  STRUCT
   FC1_SEND_1 : ARRAY  [0 .. 699 ] OF BYTE  := B#16#0;
  END_STRUCT ;
BEGIN
   FC1_SEND_1[0] := B#16#0;
   FC1_SEND_1[1] := B#16#0;
   FC1_SEND_1[2] := B#16#0;
   FC1_SEND_1[3] := B#16#0;
   FC1_SEND_1[4] := B#16#0;
   FC1_SEND_1[5] := B#16#0;
   FC1_SEND_1[6] := B#16#0;
   FC1_SEND_1[7] := B#16#0;
   FC1_SEND_1[8] := B#16#0;
   FC1_SEND_1[9] := B#16#0;
   FC1_SEND_1[10] := B#16#0;
   FC1_SEND_1[11] := B#16#0;
   FC1_SEND_1[12] := B#16#0;
   FC1_SEND_1[13] := B#16#0;
   FC1_SEND_1[14] := B#16#0;
   FC1_SEND_1[15] := B#16#0;
   FC1_SEND_1[16] := B#16#0;
   FC1_SEND_1[17] := B#16#0;
   FC1_SEND_1[18] := B#16#0;
   FC1_SEND_1[19] := B#16#0;
   FC1_SEND_1[20] := B#16#0;
   FC1_SEND_1[21] := B#16#0;
   FC1_SEND_1[22] := B#16#0;
   FC1_SEND_1[23] := B#16#0;
   FC1_SEND_1[24] := B#16#0;
   FC1_SEND_1[25] := B#16#0;
   FC1_SEND_1[26] := B#16#0;
   FC1_SEND_1[27] := B#16#0;
   FC1_SEND_1[28] := B#16#0;
   FC1_SEND_1[29] := B#16#0;
   FC1_SEND_1[30] := B#16#0;
   FC1_SEND_1[31] := B#16#0;
   FC1_SEND_1[32] := B#16#0;
   FC1_SEND_1[33] := B#16#0;
   FC1_SEND_1[34] := B#16#0;
   FC1_SEND_1[35] := B#16#0;
   FC1_SEND_1[36] := B#16#0;
   FC1_SEND_1[37] := B#16#0;
   FC1_SEND_1[38] := B#16#0;
   FC1_SEND_1[39] := B#16#0;
   FC1_SEND_1[40] := B#16#0;
   FC1_SEND_1[41] := B#16#0;
   FC1_SEND_1[42] := B#16#0;
   FC1_SEND_1[43] := B#16#0;
   FC1_SEND_1[44] := B#16#0;
   FC1_SEND_1[45] := B#16#0;
   FC1_SEND_1[46] := B#16#0;
   FC1_SEND_1[47] := B#16#0;
   FC1_SEND_1[48] := B#16#0;
   FC1_SEND_1[49] := B#16#0;
   FC1_SEND_1[50] := B#16#0;
   FC1_SEND_1[51] := B#16#0;
   FC1_SEND_1[52] := B#16#0;
   FC1_SEND_1[53] := B#16#0;
   FC1_SEND_1[54] := B#16#0;
   FC1_SEND_1[55] := B#16#0;
   FC1_SEND_1[56] := B#16#0;
   FC1_SEND_1[57] := B#16#0;
   FC1_SEND_1[58] := B#16#0;
   FC1_SEND_1[59] := B#16#0;
   FC1_SEND_1[60] := B#16#0;
   FC1_SEND_1[61] := B#16#0;
   FC1_SEND_1[62] := B#16#0;
   FC1_SEND_1[63] := B#16#0;
   FC1_SEND_1[64] := B#16#0;
   FC1_SEND_1[65] := B#16#0;
   FC1_SEND_1[66] := B#16#0;
   FC1_SEND_1[67] := B#16#0;
   FC1_SEND_1[68] := B#16#0;
   FC1_SEND_1[69] := B#16#0;
   FC1_SEND_1[70] := B#16#0;
   FC1_SEND_1[71] := B#16#0;
   FC1_SEND_1[72] := B#16#0;
   FC1_SEND_1[73] := B#16#0;
   FC1_SEND_1[74] := B#16#0;
   FC1_SEND_1[75] := B#16#0;
   FC1_SEND_1[76] := B#16#0;
   FC1_SEND_1[77] := B#16#0;
   FC1_SEND_1[78] := B#16#0;
   FC1_SEND_1[79] := B#16#0;
   FC1_SEND_1[80] := B#16#0;
   FC1_SEND_1[81] := B#16#0;
   FC1_SEND_1[82] := B#16#0;
   FC1_SEND_1[83] := B#16#0;
   FC1_SEND_1[84] := B#16#0;
   FC1_SEND_1[85] := B#16#0;
   FC1_SEND_1[86] := B#16#0;
   FC1_SEND_1[87] := B#16#0;
   FC1_SEND_1[88] := B#16#0;
   FC1_SEND_1[89] := B#16#0;
   FC1_SEND_1[90] := B#16#0;
   FC1_SEND_1[91] := B#16#0;
   FC1_SEND_1[92] := B#16#0;
   FC1_SEND_1[93] := B#16#0;
   FC1_SEND_1[94] := B#16#0;
   FC1_SEND_1[95] := B#16#0;
   FC1_SEND_1[96] := B#16#0;
   FC1_SEND_1[97] := B#16#0;
   FC1_SEND_1[98] := B#16#0;
   FC1_SEND_1[99] := B#16#0;
   FC1_SEND_1[100] := B#16#0;
   FC1_SEND_1[101] := B#16#0;
   FC1_SEND_1[102] := B#16#0;
   FC1_SEND_1[103] := B#16#0;
   FC1_SEND_1[104] := B#16#0;
   FC1_SEND_1[105] := B#16#0;
   FC1_SEND_1[106] := B#16#0;
   FC1_SEND_1[107] := B#16#0;
   FC1_SEND_1[108] := B#16#0;
   FC1_SEND_1[109] := B#16#0;
   FC1_SEND_1[110] := B#16#0;
   FC1_SEND_1[111] := B#16#0;
   FC1_SEND_1[112] := B#16#0;
   FC1_SEND_1[113] := B#16#0;
   FC1_SEND_1[114] := B#16#0;
   FC1_SEND_1[115] := B#16#0;
   FC1_SEND_1[116] := B#16#0;
   FC1_SEND_1[117] := B#16#0;
   FC1_SEND_1[118] := B#16#0;
   FC1_SEND_1[119] := B#16#0;
   FC1_SEND_1[120] := B#16#0;
   FC1_SEND_1[121] := B#16#0;
   FC1_SEND_1[122] := B#16#0;
   FC1_SEND_1[123] := B#16#0;
   FC1_SEND_1[124] := B#16#0;
   FC1_SEND_1[125] := B#16#0;
   FC1_SEND_1[126] := B#16#0;
   FC1_SEND_1[127] := B#16#0;
   FC1_SEND_1[128] := B#16#0;
   FC1_SEND_1[129] := B#16#0;
   FC1_SEND_1[130] := B#16#0;
   FC1_SEND_1[131] := B#16#0;
   FC1_SEND_1[132] := B#16#0;
   FC1_SEND_1[133] := B#16#0;
   FC1_SEND_1[134] := B#16#0;
   FC1_SEND_1[135] := B#16#0;
   FC1_SEND_1[136] := B#16#0;
   FC1_SEND_1[137] := B#16#0;
   FC1_SEND_1[138] := B#16#0;
   FC1_SEND_1[139] := B#16#0;
   FC1_SEND_1[140] := B#16#0;
   FC1_SEND_1[141] := B#16#0;
   FC1_SEND_1[142] := B#16#0;
   FC1_SEND_1[143] := B#16#0;
   FC1_SEND_1[144] := B#16#0;
   FC1_SEND_1[145] := B#16#0;
   FC1_SEND_1[146] := B#16#0;
   FC1_SEND_1[147] := B#16#0;
   FC1_SEND_1[148] := B#16#0;
   FC1_SEND_1[149] := B#16#0;
   FC1_SEND_1[150] := B#16#0;
   FC1_SEND_1[151] := B#16#0;
   FC1_SEND_1[152] := B#16#0;
   FC1_SEND_1[153] := B#16#0;
   FC1_SEND_1[154] := B#16#0;
   FC1_SEND_1[155] := B#16#0;
   FC1_SEND_1[156] := B#16#0;
   FC1_SEND_1[157] := B#16#0;
   FC1_SEND_1[158] := B#16#0;
   FC1_SEND_1[159] := B#16#0;
   FC1_SEND_1[160] := B#16#0;
   FC1_SEND_1[161] := B#16#0;
   FC1_SEND_1[162] := B#16#0;
   FC1_SEND_1[163] := B#16#0;
   FC1_SEND_1[164] := B#16#0;
   FC1_SEND_1[165] := B#16#0;
   FC1_SEND_1[166] := B#16#0;
   FC1_SEND_1[167] := B#16#0;
   FC1_SEND_1[168] := B#16#0;
   FC1_SEND_1[169] := B#16#0;
   FC1_SEND_1[170] := B#16#0;
   FC1_SEND_1[171] := B#16#0;
   FC1_SEND_1[172] := B#16#0;
   FC1_SEND_1[173] := B#16#0;
   FC1_SEND_1[174] := B#16#0;
   FC1_SEND_1[175] := B#16#0;
   FC1_SEND_1[176] := B#16#0;
   FC1_SEND_1[177] := B#16#0;
   FC1_SEND_1[178] := B#16#0;
   FC1_SEND_1[179] := B#16#0;
   FC1_SEND_1[180] := B#16#0;
   FC1_SEND_1[181] := B#16#0;
   FC1_SEND_1[182] := B#16#0;
   FC1_SEND_1[183] := B#16#0;
   FC1_SEND_1[184] := B#16#0;
   FC1_SEND_1[185] := B#16#0;
   FC1_SEND_1[186] := B#16#0;
   FC1_SEND_1[187] := B#16#0;
   FC1_SEND_1[188] := B#16#0;
   FC1_SEND_1[189] := B#16#0;
   FC1_SEND_1[190] := B#16#0;
   FC1_SEND_1[191] := B#16#0;
   FC1_SEND_1[192] := B#16#0;
   FC1_SEND_1[193] := B#16#0;
   FC1_SEND_1[194] := B#16#0;
   FC1_SEND_1[195] := B#16#0;
   FC1_SEND_1[196] := B#16#0;
   FC1_SEND_1[197] := B#16#0;
   FC1_SEND_1[198] := B#16#0;
   FC1_SEND_1[199] := B#16#0;
   FC1_SEND_1[200] := B#16#0;
   FC1_SEND_1[201] := B#16#0;
   FC1_SEND_1[202] := B#16#0;
   FC1_SEND_1[203] := B#16#0;
   FC1_SEND_1[204] := B#16#0;
   FC1_SEND_1[205] := B#16#0;
   FC1_SEND_1[206] := B#16#0;
   FC1_SEND_1[207] := B#16#0;
   FC1_SEND_1[208] := B#16#0;
   FC1_SEND_1[209] := B#16#0;
   FC1_SEND_1[210] := B#16#0;
   FC1_SEND_1[211] := B#16#0;
   FC1_SEND_1[212] := B#16#0;
   FC1_SEND_1[213] := B#16#0;
   FC1_SEND_1[214] := B#16#0;
   FC1_SEND_1[215] := B#16#0;
   FC1_SEND_1[216] := B#16#0;
   FC1_SEND_1[217] := B#16#0;
   FC1_SEND_1[218] := B#16#0;
   FC1_SEND_1[219] := B#16#0;
   FC1_SEND_1[220] := B#16#0;
   FC1_SEND_1[221] := B#16#0;
   FC1_SEND_1[222] := B#16#0;
   FC1_SEND_1[223] := B#16#0;
   FC1_SEND_1[224] := B#16#0;
   FC1_SEND_1[225] := B#16#0;
   FC1_SEND_1[226] := B#16#0;
   FC1_SEND_1[227] := B#16#0;
   FC1_SEND_1[228] := B#16#0;
   FC1_SEND_1[229] := B#16#0;
   FC1_SEND_1[230] := B#16#0;
   FC1_SEND_1[231] := B#16#0;
   FC1_SEND_1[232] := B#16#0;
   FC1_SEND_1[233] := B#16#0;
   FC1_SEND_1[234] := B#16#0;
   FC1_SEND_1[235] := B#16#0;
   FC1_SEND_1[236] := B#16#0;
   FC1_SEND_1[237] := B#16#0;
   FC1_SEND_1[238] := B#16#0;
   FC1_SEND_1[239] := B#16#0;
   FC1_SEND_1[240] := B#16#0;
   FC1_SEND_1[241] := B#16#0;
   FC1_SEND_1[242] := B#16#0;
   FC1_SEND_1[243] := B#16#0;
   FC1_SEND_1[244] := B#16#0;
   FC1_SEND_1[245] := B#16#0;
   FC1_SEND_1[246] := B#16#0;
   FC1_SEND_1[247] := B#16#0;
   FC1_SEND_1[248] := B#16#0;
   FC1_SEND_1[249] := B#16#0;
   FC1_SEND_1[250] := B#16#0;
   FC1_SEND_1[251] := B#16#0;
   FC1_SEND_1[252] := B#16#0;
   FC1_SEND_1[253] := B#16#0;
   FC1_SEND_1[254] := B#16#0;
   FC1_SEND_1[255] := B#16#0;
   FC1_SEND_1[256] := B#16#0;
   FC1_SEND_1[257] := B#16#0;
   FC1_SEND_1[258] := B#16#0;
   FC1_SEND_1[259] := B#16#0;
   FC1_SEND_1[260] := B#16#0;
   FC1_SEND_1[261] := B#16#0;
   FC1_SEND_1[262] := B#16#0;
   FC1_SEND_1[263] := B#16#0;
   FC1_SEND_1[264] := B#16#0;
   FC1_SEND_1[265] := B#16#0;
   FC1_SEND_1[266] := B#16#0;
   FC1_SEND_1[267] := B#16#0;
   FC1_SEND_1[268] := B#16#0;
   FC1_SEND_1[269] := B#16#0;
   FC1_SEND_1[270] := B#16#0;
   FC1_SEND_1[271] := B#16#0;
   FC1_SEND_1[272] := B#16#0;
   FC1_SEND_1[273] := B#16#0;
   FC1_SEND_1[274] := B#16#0;
   FC1_SEND_1[275] := B#16#0;
   FC1_SEND_1[276] := B#16#0;
   FC1_SEND_1[277] := B#16#0;
   FC1_SEND_1[278] := B#16#0;
   FC1_SEND_1[279] := B#16#0;
   FC1_SEND_1[280] := B#16#0;
   FC1_SEND_1[281] := B#16#0;
   FC1_SEND_1[282] := B#16#0;
   FC1_SEND_1[283] := B#16#0;
   FC1_SEND_1[284] := B#16#0;
   FC1_SEND_1[285] := B#16#0;
   FC1_SEND_1[286] := B#16#0;
   FC1_SEND_1[287] := B#16#0;
   FC1_SEND_1[288] := B#16#0;
   FC1_SEND_1[289] := B#16#0;
   FC1_SEND_1[290] := B#16#0;
   FC1_SEND_1[291] := B#16#0;
   FC1_SEND_1[292] := B#16#0;
   FC1_SEND_1[293] := B#16#0;
   FC1_SEND_1[294] := B#16#0;
   FC1_SEND_1[295] := B#16#0;
   FC1_SEND_1[296] := B#16#0;
   FC1_SEND_1[297] := B#16#0;
   FC1_SEND_1[298] := B#16#0;
   FC1_SEND_1[299] := B#16#0;
   FC1_SEND_1[300] := B#16#0;
   FC1_SEND_1[301] := B#16#0;
   FC1_SEND_1[302] := B#16#0;
   FC1_SEND_1[303] := B#16#0;
   FC1_SEND_1[304] := B#16#0;
   FC1_SEND_1[305] := B#16#0;
   FC1_SEND_1[306] := B#16#0;
   FC1_SEND_1[307] := B#16#0;
   FC1_SEND_1[308] := B#16#0;
   FC1_SEND_1[309] := B#16#0;
   FC1_SEND_1[310] := B#16#0;
   FC1_SEND_1[311] := B#16#0;
   FC1_SEND_1[312] := B#16#0;
   FC1_SEND_1[313] := B#16#0;
   FC1_SEND_1[314] := B#16#0;
   FC1_SEND_1[315] := B#16#0;
   FC1_SEND_1[316] := B#16#0;
   FC1_SEND_1[317] := B#16#0;
   FC1_SEND_1[318] := B#16#0;
   FC1_SEND_1[319] := B#16#0;
   FC1_SEND_1[320] := B#16#0;
   FC1_SEND_1[321] := B#16#0;
   FC1_SEND_1[322] := B#16#0;
   FC1_SEND_1[323] := B#16#0;
   FC1_SEND_1[324] := B#16#0;
   FC1_SEND_1[325] := B#16#0;
   FC1_SEND_1[326] := B#16#0;
   FC1_SEND_1[327] := B#16#0;
   FC1_SEND_1[328] := B#16#0;
   FC1_SEND_1[329] := B#16#0;
   FC1_SEND_1[330] := B#16#0;
   FC1_SEND_1[331] := B#16#0;
   FC1_SEND_1[332] := B#16#0;
   FC1_SEND_1[333] := B#16#0;
   FC1_SEND_1[334] := B#16#0;
   FC1_SEND_1[335] := B#16#0;
   FC1_SEND_1[336] := B#16#0;
   FC1_SEND_1[337] := B#16#0;
   FC1_SEND_1[338] := B#16#0;
   FC1_SEND_1[339] := B#16#0;
   FC1_SEND_1[340] := B#16#0;
   FC1_SEND_1[341] := B#16#0;
   FC1_SEND_1[342] := B#16#0;
   FC1_SEND_1[343] := B#16#0;
   FC1_SEND_1[344] := B#16#0;
   FC1_SEND_1[345] := B#16#0;
   FC1_SEND_1[346] := B#16#0;
   FC1_SEND_1[347] := B#16#0;
   FC1_SEND_1[348] := B#16#0;
   FC1_SEND_1[349] := B#16#0;
   FC1_SEND_1[350] := B#16#0;
   FC1_SEND_1[351] := B#16#0;
   FC1_SEND_1[352] := B#16#0;
   FC1_SEND_1[353] := B#16#0;
   FC1_SEND_1[354] := B#16#0;
   FC1_SEND_1[355] := B#16#0;
   FC1_SEND_1[356] := B#16#0;
   FC1_SEND_1[357] := B#16#0;
   FC1_SEND_1[358] := B#16#0;
   FC1_SEND_1[359] := B#16#0;
   FC1_SEND_1[360] := B#16#0;
   FC1_SEND_1[361] := B#16#0;
   FC1_SEND_1[362] := B#16#0;
   FC1_SEND_1[363] := B#16#0;
   FC1_SEND_1[364] := B#16#0;
   FC1_SEND_1[365] := B#16#0;
   FC1_SEND_1[366] := B#16#0;
   FC1_SEND_1[367] := B#16#0;
   FC1_SEND_1[368] := B#16#0;
   FC1_SEND_1[369] := B#16#0;
   FC1_SEND_1[370] := B#16#0;
   FC1_SEND_1[371] := B#16#0;
   FC1_SEND_1[372] := B#16#0;
   FC1_SEND_1[373] := B#16#0;
   FC1_SEND_1[374] := B#16#0;
   FC1_SEND_1[375] := B#16#0;
   FC1_SEND_1[376] := B#16#0;
   FC1_SEND_1[377] := B#16#0;
   FC1_SEND_1[378] := B#16#0;
   FC1_SEND_1[379] := B#16#0;
   FC1_SEND_1[380] := B#16#0;
   FC1_SEND_1[381] := B#16#0;
   FC1_SEND_1[382] := B#16#0;
   FC1_SEND_1[383] := B#16#0;
   FC1_SEND_1[384] := B#16#0;
   FC1_SEND_1[385] := B#16#0;
   FC1_SEND_1[386] := B#16#0;
   FC1_SEND_1[387] := B#16#0;
   FC1_SEND_1[388] := B#16#0;
   FC1_SEND_1[389] := B#16#0;
   FC1_SEND_1[390] := B#16#0;
   FC1_SEND_1[391] := B#16#0;
   FC1_SEND_1[392] := B#16#0;
   FC1_SEND_1[393] := B#16#0;
   FC1_SEND_1[394] := B#16#0;
   FC1_SEND_1[395] := B#16#0;
   FC1_SEND_1[396] := B#16#0;
   FC1_SEND_1[397] := B#16#0;
   FC1_SEND_1[398] := B#16#0;
   FC1_SEND_1[399] := B#16#0;
   FC1_SEND_1[400] := B#16#0;
   FC1_SEND_1[401] := B#16#0;
   FC1_SEND_1[402] := B#16#0;
   FC1_SEND_1[403] := B#16#0;
   FC1_SEND_1[404] := B#16#0;
   FC1_SEND_1[405] := B#16#0;
   FC1_SEND_1[406] := B#16#0;
   FC1_SEND_1[407] := B#16#0;
   FC1_SEND_1[408] := B#16#0;
   FC1_SEND_1[409] := B#16#0;
   FC1_SEND_1[410] := B#16#0;
   FC1_SEND_1[411] := B#16#0;
   FC1_SEND_1[412] := B#16#0;
   FC1_SEND_1[413] := B#16#0;
   FC1_SEND_1[414] := B#16#0;
   FC1_SEND_1[415] := B#16#0;
   FC1_SEND_1[416] := B#16#0;
   FC1_SEND_1[417] := B#16#0;
   FC1_SEND_1[418] := B#16#0;
   FC1_SEND_1[419] := B#16#0;
   FC1_SEND_1[420] := B#16#0;
   FC1_SEND_1[421] := B#16#0;
   FC1_SEND_1[422] := B#16#0;
   FC1_SEND_1[423] := B#16#0;
   FC1_SEND_1[424] := B#16#0;
   FC1_SEND_1[425] := B#16#0;
   FC1_SEND_1[426] := B#16#0;
   FC1_SEND_1[427] := B#16#0;
   FC1_SEND_1[428] := B#16#0;
   FC1_SEND_1[429] := B#16#0;
   FC1_SEND_1[430] := B#16#0;
   FC1_SEND_1[431] := B#16#0;
   FC1_SEND_1[432] := B#16#0;
   FC1_SEND_1[433] := B#16#0;
   FC1_SEND_1[434] := B#16#0;
   FC1_SEND_1[435] := B#16#0;
   FC1_SEND_1[436] := B#16#0;
   FC1_SEND_1[437] := B#16#0;
   FC1_SEND_1[438] := B#16#0;
   FC1_SEND_1[439] := B#16#0;
   FC1_SEND_1[440] := B#16#0;
   FC1_SEND_1[441] := B#16#0;
   FC1_SEND_1[442] := B#16#0;
   FC1_SEND_1[443] := B#16#0;
   FC1_SEND_1[444] := B#16#0;
   FC1_SEND_1[445] := B#16#0;
   FC1_SEND_1[446] := B#16#0;
   FC1_SEND_1[447] := B#16#0;
   FC1_SEND_1[448] := B#16#0;
   FC1_SEND_1[449] := B#16#0;
   FC1_SEND_1[450] := B#16#0;
   FC1_SEND_1[451] := B#16#0;
   FC1_SEND_1[452] := B#16#0;
   FC1_SEND_1[453] := B#16#0;
   FC1_SEND_1[454] := B#16#0;
   FC1_SEND_1[455] := B#16#0;
   FC1_SEND_1[456] := B#16#0;
   FC1_SEND_1[457] := B#16#0;
   FC1_SEND_1[458] := B#16#0;
   FC1_SEND_1[459] := B#16#0;
   FC1_SEND_1[460] := B#16#0;
   FC1_SEND_1[461] := B#16#0;
   FC1_SEND_1[462] := B#16#0;
   FC1_SEND_1[463] := B#16#0;
   FC1_SEND_1[464] := B#16#0;
   FC1_SEND_1[465] := B#16#0;
   FC1_SEND_1[466] := B#16#0;
   FC1_SEND_1[467] := B#16#0;
   FC1_SEND_1[468] := B#16#0;
   FC1_SEND_1[469] := B#16#0;
   FC1_SEND_1[470] := B#16#0;
   FC1_SEND_1[471] := B#16#0;
   FC1_SEND_1[472] := B#16#0;
   FC1_SEND_1[473] := B#16#0;
   FC1_SEND_1[474] := B#16#0;
   FC1_SEND_1[475] := B#16#0;
   FC1_SEND_1[476] := B#16#0;
   FC1_SEND_1[477] := B#16#0;
   FC1_SEND_1[478] := B#16#0;
   FC1_SEND_1[479] := B#16#0;
   FC1_SEND_1[480] := B#16#0;
   FC1_SEND_1[481] := B#16#0;
   FC1_SEND_1[482] := B#16#0;
   FC1_SEND_1[483] := B#16#0;
   FC1_SEND_1[484] := B#16#0;
   FC1_SEND_1[485] := B#16#0;
   FC1_SEND_1[486] := B#16#0;
   FC1_SEND_1[487] := B#16#0;
   FC1_SEND_1[488] := B#16#0;
   FC1_SEND_1[489] := B#16#0;
   FC1_SEND_1[490] := B#16#0;
   FC1_SEND_1[491] := B#16#0;
   FC1_SEND_1[492] := B#16#0;
   FC1_SEND_1[493] := B#16#0;
   FC1_SEND_1[494] := B#16#0;
   FC1_SEND_1[495] := B#16#0;
   FC1_SEND_1[496] := B#16#0;
   FC1_SEND_1[497] := B#16#0;
   FC1_SEND_1[498] := B#16#0;
   FC1_SEND_1[499] := B#16#0;
   FC1_SEND_1[500] := B#16#0;
   FC1_SEND_1[501] := B#16#0;
   FC1_SEND_1[502] := B#16#0;
   FC1_SEND_1[503] := B#16#0;
   FC1_SEND_1[504] := B#16#0;
   FC1_SEND_1[505] := B#16#0;
   FC1_SEND_1[506] := B#16#0;
   FC1_SEND_1[507] := B#16#0;
   FC1_SEND_1[508] := B#16#0;
   FC1_SEND_1[509] := B#16#0;
   FC1_SEND_1[510] := B#16#0;
   FC1_SEND_1[511] := B#16#0;
   FC1_SEND_1[512] := B#16#0;
   FC1_SEND_1[513] := B#16#0;
   FC1_SEND_1[514] := B#16#0;
   FC1_SEND_1[515] := B#16#0;
   FC1_SEND_1[516] := B#16#0;
   FC1_SEND_1[517] := B#16#0;
   FC1_SEND_1[518] := B#16#0;
   FC1_SEND_1[519] := B#16#0;
   FC1_SEND_1[520] := B#16#0;
   FC1_SEND_1[521] := B#16#0;
   FC1_SEND_1[522] := B#16#0;
   FC1_SEND_1[523] := B#16#0;
   FC1_SEND_1[524] := B#16#0;
   FC1_SEND_1[525] := B#16#0;
   FC1_SEND_1[526] := B#16#0;
   FC1_SEND_1[527] := B#16#0;
   FC1_SEND_1[528] := B#16#0;
   FC1_SEND_1[529] := B#16#0;
   FC1_SEND_1[530] := B#16#0;
   FC1_SEND_1[531] := B#16#0;
   FC1_SEND_1[532] := B#16#0;
   FC1_SEND_1[533] := B#16#0;
   FC1_SEND_1[534] := B#16#0;
   FC1_SEND_1[535] := B#16#0;
   FC1_SEND_1[536] := B#16#0;
   FC1_SEND_1[537] := B#16#0;
   FC1_SEND_1[538] := B#16#0;
   FC1_SEND_1[539] := B#16#0;
   FC1_SEND_1[540] := B#16#0;
   FC1_SEND_1[541] := B#16#0;
   FC1_SEND_1[542] := B#16#0;
   FC1_SEND_1[543] := B#16#0;
   FC1_SEND_1[544] := B#16#0;
   FC1_SEND_1[545] := B#16#0;
   FC1_SEND_1[546] := B#16#0;
   FC1_SEND_1[547] := B#16#0;
   FC1_SEND_1[548] := B#16#0;
   FC1_SEND_1[549] := B#16#0;
   FC1_SEND_1[550] := B#16#0;
   FC1_SEND_1[551] := B#16#0;
   FC1_SEND_1[552] := B#16#0;
   FC1_SEND_1[553] := B#16#0;
   FC1_SEND_1[554] := B#16#0;
   FC1_SEND_1[555] := B#16#0;
   FC1_SEND_1[556] := B#16#0;
   FC1_SEND_1[557] := B#16#0;
   FC1_SEND_1[558] := B#16#0;
   FC1_SEND_1[559] := B#16#0;
   FC1_SEND_1[560] := B#16#0;
   FC1_SEND_1[561] := B#16#0;
   FC1_SEND_1[562] := B#16#0;
   FC1_SEND_1[563] := B#16#0;
   FC1_SEND_1[564] := B#16#0;
   FC1_SEND_1[565] := B#16#0;
   FC1_SEND_1[566] := B#16#0;
   FC1_SEND_1[567] := B#16#0;
   FC1_SEND_1[568] := B#16#0;
   FC1_SEND_1[569] := B#16#0;
   FC1_SEND_1[570] := B#16#0;
   FC1_SEND_1[571] := B#16#0;
   FC1_SEND_1[572] := B#16#0;
   FC1_SEND_1[573] := B#16#0;
   FC1_SEND_1[574] := B#16#0;
   FC1_SEND_1[575] := B#16#0;
   FC1_SEND_1[576] := B#16#0;
   FC1_SEND_1[577] := B#16#0;
   FC1_SEND_1[578] := B#16#0;
   FC1_SEND_1[579] := B#16#0;
   FC1_SEND_1[580] := B#16#0;
   FC1_SEND_1[581] := B#16#0;
   FC1_SEND_1[582] := B#16#0;
   FC1_SEND_1[583] := B#16#0;
   FC1_SEND_1[584] := B#16#0;
   FC1_SEND_1[585] := B#16#0;
   FC1_SEND_1[586] := B#16#0;
   FC1_SEND_1[587] := B#16#0;
   FC1_SEND_1[588] := B#16#0;
   FC1_SEND_1[589] := B#16#0;
   FC1_SEND_1[590] := B#16#0;
   FC1_SEND_1[591] := B#16#0;
   FC1_SEND_1[592] := B#16#0;
   FC1_SEND_1[593] := B#16#0;
   FC1_SEND_1[594] := B#16#0;
   FC1_SEND_1[595] := B#16#0;
   FC1_SEND_1[596] := B#16#0;
   FC1_SEND_1[597] := B#16#0;
   FC1_SEND_1[598] := B#16#0;
   FC1_SEND_1[599] := B#16#0;
   FC1_SEND_1[600] := B#16#0;
   FC1_SEND_1[601] := B#16#0;
   FC1_SEND_1[602] := B#16#0;
   FC1_SEND_1[603] := B#16#0;
   FC1_SEND_1[604] := B#16#0;
   FC1_SEND_1[605] := B#16#0;
   FC1_SEND_1[606] := B#16#0;
   FC1_SEND_1[607] := B#16#0;
   FC1_SEND_1[608] := B#16#0;
   FC1_SEND_1[609] := B#16#0;
   FC1_SEND_1[610] := B#16#0;
   FC1_SEND_1[611] := B#16#0;
   FC1_SEND_1[612] := B#16#0;
   FC1_SEND_1[613] := B#16#0;
   FC1_SEND_1[614] := B#16#0;
   FC1_SEND_1[615] := B#16#0;
   FC1_SEND_1[616] := B#16#0;
   FC1_SEND_1[617] := B#16#0;
   FC1_SEND_1[618] := B#16#0;
   FC1_SEND_1[619] := B#16#0;
   FC1_SEND_1[620] := B#16#0;
   FC1_SEND_1[621] := B#16#0;
   FC1_SEND_1[622] := B#16#0;
   FC1_SEND_1[623] := B#16#0;
   FC1_SEND_1[624] := B#16#0;
   FC1_SEND_1[625] := B#16#0;
   FC1_SEND_1[626] := B#16#0;
   FC1_SEND_1[627] := B#16#0;
   FC1_SEND_1[628] := B#16#0;
   FC1_SEND_1[629] := B#16#0;
   FC1_SEND_1[630] := B#16#0;
   FC1_SEND_1[631] := B#16#0;
   FC1_SEND_1[632] := B#16#0;
   FC1_SEND_1[633] := B#16#0;
   FC1_SEND_1[634] := B#16#0;
   FC1_SEND_1[635] := B#16#0;
   FC1_SEND_1[636] := B#16#0;
   FC1_SEND_1[637] := B#16#0;
   FC1_SEND_1[638] := B#16#0;
   FC1_SEND_1[639] := B#16#0;
   FC1_SEND_1[640] := B#16#0;
   FC1_SEND_1[641] := B#16#0;
   FC1_SEND_1[642] := B#16#0;
   FC1_SEND_1[643] := B#16#0;
   FC1_SEND_1[644] := B#16#0;
   FC1_SEND_1[645] := B#16#0;
   FC1_SEND_1[646] := B#16#0;
   FC1_SEND_1[647] := B#16#0;
   FC1_SEND_1[648] := B#16#0;
   FC1_SEND_1[649] := B#16#0;
   FC1_SEND_1[650] := B#16#0;
   FC1_SEND_1[651] := B#16#0;
   FC1_SEND_1[652] := B#16#0;
   FC1_SEND_1[653] := B#16#0;
   FC1_SEND_1[654] := B#16#0;
   FC1_SEND_1[655] := B#16#0;
   FC1_SEND_1[656] := B#16#0;
   FC1_SEND_1[657] := B#16#0;
   FC1_SEND_1[658] := B#16#0;
   FC1_SEND_1[659] := B#16#0;
   FC1_SEND_1[660] := B#16#0;
   FC1_SEND_1[661] := B#16#0;
   FC1_SEND_1[662] := B#16#0;
   FC1_SEND_1[663] := B#16#0;
   FC1_SEND_1[664] := B#16#0;
   FC1_SEND_1[665] := B#16#0;
   FC1_SEND_1[666] := B#16#0;
   FC1_SEND_1[667] := B#16#0;
   FC1_SEND_1[668] := B#16#0;
   FC1_SEND_1[669] := B#16#0;
   FC1_SEND_1[670] := B#16#0;
   FC1_SEND_1[671] := B#16#0;
   FC1_SEND_1[672] := B#16#0;
   FC1_SEND_1[673] := B#16#0;
   FC1_SEND_1[674] := B#16#0;
   FC1_SEND_1[675] := B#16#0;
   FC1_SEND_1[676] := B#16#0;
   FC1_SEND_1[677] := B#16#0;
   FC1_SEND_1[678] := B#16#0;
   FC1_SEND_1[679] := B#16#0;
   FC1_SEND_1[680] := B#16#0;
   FC1_SEND_1[681] := B#16#0;
   FC1_SEND_1[682] := B#16#0;
   FC1_SEND_1[683] := B#16#0;
   FC1_SEND_1[684] := B#16#0;
   FC1_SEND_1[685] := B#16#0;
   FC1_SEND_1[686] := B#16#0;
   FC1_SEND_1[687] := B#16#0;
   FC1_SEND_1[688] := B#16#0;
   FC1_SEND_1[689] := B#16#0;
   FC1_SEND_1[690] := B#16#0;
   FC1_SEND_1[691] := B#16#0;
   FC1_SEND_1[692] := B#16#0;
   FC1_SEND_1[693] := B#16#0;
   FC1_SEND_1[694] := B#16#0;
   FC1_SEND_1[695] := B#16#0;
   FC1_SEND_1[696] := B#16#0;
   FC1_SEND_1[697] := B#16#0;
   FC1_SEND_1[698] := B#16#0;
   FC1_SEND_1[699] := B#16#0;
END_DATA_BLOCK

DATA_BLOCK DB 61
TITLE =
VERSION : 0.1


  STRUCT
   FC2_RECV_1 : ARRAY  [0 .. 699 ] OF BYTE  := B#16#0;
  END_STRUCT ;
BEGIN
   FC2_RECV_1[0] := B#16#0;
   FC2_RECV_1[1] := B#16#0;
   FC2_RECV_1[2] := B#16#0;
   FC2_RECV_1[3] := B#16#0;
   FC2_RECV_1[4] := B#16#0;
   FC2_RECV_1[5] := B#16#0;
   FC2_RECV_1[6] := B#16#0;
   FC2_RECV_1[7] := B#16#0;
   FC2_RECV_1[8] := B#16#0;
   FC2_RECV_1[9] := B#16#0;
   FC2_RECV_1[10] := B#16#0;
   FC2_RECV_1[11] := B#16#0;
   FC2_RECV_1[12] := B#16#0;
   FC2_RECV_1[13] := B#16#0;
   FC2_RECV_1[14] := B#16#0;
   FC2_RECV_1[15] := B#16#0;
   FC2_RECV_1[16] := B#16#0;
   FC2_RECV_1[17] := B#16#0;
   FC2_RECV_1[18] := B#16#0;
   FC2_RECV_1[19] := B#16#0;
   FC2_RECV_1[20] := B#16#0;
   FC2_RECV_1[21] := B#16#0;
   FC2_RECV_1[22] := B#16#0;
   FC2_RECV_1[23] := B#16#0;
   FC2_RECV_1[24] := B#16#0;
   FC2_RECV_1[25] := B#16#0;
   FC2_RECV_1[26] := B#16#0;
   FC2_RECV_1[27] := B#16#0;
   FC2_RECV_1[28] := B#16#0;
   FC2_RECV_1[29] := B#16#0;
   FC2_RECV_1[30] := B#16#0;
   FC2_RECV_1[31] := B#16#0;
   FC2_RECV_1[32] := B#16#0;
   FC2_RECV_1[33] := B#16#0;
   FC2_RECV_1[34] := B#16#0;
   FC2_RECV_1[35] := B#16#0;
   FC2_RECV_1[36] := B#16#0;
   FC2_RECV_1[37] := B#16#0;
   FC2_RECV_1[38] := B#16#0;
   FC2_RECV_1[39] := B#16#0;
   FC2_RECV_1[40] := B#16#0;
   FC2_RECV_1[41] := B#16#0;
   FC2_RECV_1[42] := B#16#0;
   FC2_RECV_1[43] := B#16#0;
   FC2_RECV_1[44] := B#16#0;
   FC2_RECV_1[45] := B#16#0;
   FC2_RECV_1[46] := B#16#0;
   FC2_RECV_1[47] := B#16#0;
   FC2_RECV_1[48] := B#16#0;
   FC2_RECV_1[49] := B#16#0;
   FC2_RECV_1[50] := B#16#0;
   FC2_RECV_1[51] := B#16#0;
   FC2_RECV_1[52] := B#16#0;
   FC2_RECV_1[53] := B#16#0;
   FC2_RECV_1[54] := B#16#0;
   FC2_RECV_1[55] := B#16#0;
   FC2_RECV_1[56] := B#16#0;
   FC2_RECV_1[57] := B#16#0;
   FC2_RECV_1[58] := B#16#0;
   FC2_RECV_1[59] := B#16#0;
   FC2_RECV_1[60] := B#16#0;
   FC2_RECV_1[61] := B#16#0;
   FC2_RECV_1[62] := B#16#0;
   FC2_RECV_1[63] := B#16#0;
   FC2_RECV_1[64] := B#16#0;
   FC2_RECV_1[65] := B#16#0;
   FC2_RECV_1[66] := B#16#0;
   FC2_RECV_1[67] := B#16#0;
   FC2_RECV_1[68] := B#16#0;
   FC2_RECV_1[69] := B#16#0;
   FC2_RECV_1[70] := B#16#0;
   FC2_RECV_1[71] := B#16#0;
   FC2_RECV_1[72] := B#16#0;
   FC2_RECV_1[73] := B#16#0;
   FC2_RECV_1[74] := B#16#0;
   FC2_RECV_1[75] := B#16#0;
   FC2_RECV_1[76] := B#16#0;
   FC2_RECV_1[77] := B#16#0;
   FC2_RECV_1[78] := B#16#0;
   FC2_RECV_1[79] := B#16#0;
   FC2_RECV_1[80] := B#16#0;
   FC2_RECV_1[81] := B#16#0;
   FC2_RECV_1[82] := B#16#0;
   FC2_RECV_1[83] := B#16#0;
   FC2_RECV_1[84] := B#16#0;
   FC2_RECV_1[85] := B#16#0;
   FC2_RECV_1[86] := B#16#0;
   FC2_RECV_1[87] := B#16#0;
   FC2_RECV_1[88] := B#16#0;
   FC2_RECV_1[89] := B#16#0;
   FC2_RECV_1[90] := B#16#0;
   FC2_RECV_1[91] := B#16#0;
   FC2_RECV_1[92] := B#16#0;
   FC2_RECV_1[93] := B#16#0;
   FC2_RECV_1[94] := B#16#0;
   FC2_RECV_1[95] := B#16#0;
   FC2_RECV_1[96] := B#16#0;
   FC2_RECV_1[97] := B#16#0;
   FC2_RECV_1[98] := B#16#0;
   FC2_RECV_1[99] := B#16#0;
   FC2_RECV_1[100] := B#16#0;
   FC2_RECV_1[101] := B#16#0;
   FC2_RECV_1[102] := B#16#0;
   FC2_RECV_1[103] := B#16#0;
   FC2_RECV_1[104] := B#16#0;
   FC2_RECV_1[105] := B#16#0;
   FC2_RECV_1[106] := B#16#0;
   FC2_RECV_1[107] := B#16#0;
   FC2_RECV_1[108] := B#16#0;
   FC2_RECV_1[109] := B#16#0;
   FC2_RECV_1[110] := B#16#0;
   FC2_RECV_1[111] := B#16#0;
   FC2_RECV_1[112] := B#16#0;
   FC2_RECV_1[113] := B#16#0;
   FC2_RECV_1[114] := B#16#0;
   FC2_RECV_1[115] := B#16#0;
   FC2_RECV_1[116] := B#16#0;
   FC2_RECV_1[117] := B#16#0;
   FC2_RECV_1[118] := B#16#0;
   FC2_RECV_1[119] := B#16#0;
   FC2_RECV_1[120] := B#16#0;
   FC2_RECV_1[121] := B#16#0;
   FC2_RECV_1[122] := B#16#0;
   FC2_RECV_1[123] := B#16#0;
   FC2_RECV_1[124] := B#16#0;
   FC2_RECV_1[125] := B#16#0;
   FC2_RECV_1[126] := B#16#0;
   FC2_RECV_1[127] := B#16#0;
   FC2_RECV_1[128] := B#16#0;
   FC2_RECV_1[129] := B#16#0;
   FC2_RECV_1[130] := B#16#0;
   FC2_RECV_1[131] := B#16#0;
   FC2_RECV_1[132] := B#16#0;
   FC2_RECV_1[133] := B#16#0;
   FC2_RECV_1[134] := B#16#0;
   FC2_RECV_1[135] := B#16#0;
   FC2_RECV_1[136] := B#16#0;
   FC2_RECV_1[137] := B#16#0;
   FC2_RECV_1[138] := B#16#0;
   FC2_RECV_1[139] := B#16#0;
   FC2_RECV_1[140] := B#16#0;
   FC2_RECV_1[141] := B#16#0;
   FC2_RECV_1[142] := B#16#0;
   FC2_RECV_1[143] := B#16#0;
   FC2_RECV_1[144] := B#16#0;
   FC2_RECV_1[145] := B#16#0;
   FC2_RECV_1[146] := B#16#0;
   FC2_RECV_1[147] := B#16#0;
   FC2_RECV_1[148] := B#16#0;
   FC2_RECV_1[149] := B#16#0;
   FC2_RECV_1[150] := B#16#0;
   FC2_RECV_1[151] := B#16#0;
   FC2_RECV_1[152] := B#16#0;
   FC2_RECV_1[153] := B#16#0;
   FC2_RECV_1[154] := B#16#0;
   FC2_RECV_1[155] := B#16#0;
   FC2_RECV_1[156] := B#16#0;
   FC2_RECV_1[157] := B#16#0;
   FC2_RECV_1[158] := B#16#0;
   FC2_RECV_1[159] := B#16#0;
   FC2_RECV_1[160] := B#16#0;
   FC2_RECV_1[161] := B#16#0;
   FC2_RECV_1[162] := B#16#0;
   FC2_RECV_1[163] := B#16#0;
   FC2_RECV_1[164] := B#16#0;
   FC2_RECV_1[165] := B#16#0;
   FC2_RECV_1[166] := B#16#0;
   FC2_RECV_1[167] := B#16#0;
   FC2_RECV_1[168] := B#16#0;
   FC2_RECV_1[169] := B#16#0;
   FC2_RECV_1[170] := B#16#0;
   FC2_RECV_1[171] := B#16#0;
   FC2_RECV_1[172] := B#16#0;
   FC2_RECV_1[173] := B#16#0;
   FC2_RECV_1[174] := B#16#0;
   FC2_RECV_1[175] := B#16#0;
   FC2_RECV_1[176] := B#16#0;
   FC2_RECV_1[177] := B#16#0;
   FC2_RECV_1[178] := B#16#0;
   FC2_RECV_1[179] := B#16#0;
   FC2_RECV_1[180] := B#16#0;
   FC2_RECV_1[181] := B#16#0;
   FC2_RECV_1[182] := B#16#0;
   FC2_RECV_1[183] := B#16#0;
   FC2_RECV_1[184] := B#16#0;
   FC2_RECV_1[185] := B#16#0;
   FC2_RECV_1[186] := B#16#0;
   FC2_RECV_1[187] := B#16#0;
   FC2_RECV_1[188] := B#16#0;
   FC2_RECV_1[189] := B#16#0;
   FC2_RECV_1[190] := B#16#0;
   FC2_RECV_1[191] := B#16#0;
   FC2_RECV_1[192] := B#16#0;
   FC2_RECV_1[193] := B#16#0;
   FC2_RECV_1[194] := B#16#0;
   FC2_RECV_1[195] := B#16#0;
   FC2_RECV_1[196] := B#16#0;
   FC2_RECV_1[197] := B#16#0;
   FC2_RECV_1[198] := B#16#0;
   FC2_RECV_1[199] := B#16#0;
   FC2_RECV_1[200] := B#16#0;
   FC2_RECV_1[201] := B#16#0;
   FC2_RECV_1[202] := B#16#0;
   FC2_RECV_1[203] := B#16#0;
   FC2_RECV_1[204] := B#16#0;
   FC2_RECV_1[205] := B#16#0;
   FC2_RECV_1[206] := B#16#0;
   FC2_RECV_1[207] := B#16#0;
   FC2_RECV_1[208] := B#16#0;
   FC2_RECV_1[209] := B#16#0;
   FC2_RECV_1[210] := B#16#0;
   FC2_RECV_1[211] := B#16#0;
   FC2_RECV_1[212] := B#16#0;
   FC2_RECV_1[213] := B#16#0;
   FC2_RECV_1[214] := B#16#0;
   FC2_RECV_1[215] := B#16#0;
   FC2_RECV_1[216] := B#16#0;
   FC2_RECV_1[217] := B#16#0;
   FC2_RECV_1[218] := B#16#0;
   FC2_RECV_1[219] := B#16#0;
   FC2_RECV_1[220] := B#16#0;
   FC2_RECV_1[221] := B#16#0;
   FC2_RECV_1[222] := B#16#0;
   FC2_RECV_1[223] := B#16#0;
   FC2_RECV_1[224] := B#16#0;
   FC2_RECV_1[225] := B#16#0;
   FC2_RECV_1[226] := B#16#0;
   FC2_RECV_1[227] := B#16#0;
   FC2_RECV_1[228] := B#16#0;
   FC2_RECV_1[229] := B#16#0;
   FC2_RECV_1[230] := B#16#0;
   FC2_RECV_1[231] := B#16#0;
   FC2_RECV_1[232] := B#16#0;
   FC2_RECV_1[233] := B#16#0;
   FC2_RECV_1[234] := B#16#0;
   FC2_RECV_1[235] := B#16#0;
   FC2_RECV_1[236] := B#16#0;
   FC2_RECV_1[237] := B#16#0;
   FC2_RECV_1[238] := B#16#0;
   FC2_RECV_1[239] := B#16#0;
   FC2_RECV_1[240] := B#16#0;
   FC2_RECV_1[241] := B#16#0;
   FC2_RECV_1[242] := B#16#0;
   FC2_RECV_1[243] := B#16#0;
   FC2_RECV_1[244] := B#16#0;
   FC2_RECV_1[245] := B#16#0;
   FC2_RECV_1[246] := B#16#0;
   FC2_RECV_1[247] := B#16#0;
   FC2_RECV_1[248] := B#16#0;
   FC2_RECV_1[249] := B#16#0;
   FC2_RECV_1[250] := B#16#0;
   FC2_RECV_1[251] := B#16#0;
   FC2_RECV_1[252] := B#16#0;
   FC2_RECV_1[253] := B#16#0;
   FC2_RECV_1[254] := B#16#0;
   FC2_RECV_1[255] := B#16#0;
   FC2_RECV_1[256] := B#16#0;
   FC2_RECV_1[257] := B#16#0;
   FC2_RECV_1[258] := B#16#0;
   FC2_RECV_1[259] := B#16#0;
   FC2_RECV_1[260] := B#16#0;
   FC2_RECV_1[261] := B#16#0;
   FC2_RECV_1[262] := B#16#0;
   FC2_RECV_1[263] := B#16#0;
   FC2_RECV_1[264] := B#16#0;
   FC2_RECV_1[265] := B#16#0;
   FC2_RECV_1[266] := B#16#0;
   FC2_RECV_1[267] := B#16#0;
   FC2_RECV_1[268] := B#16#0;
   FC2_RECV_1[269] := B#16#0;
   FC2_RECV_1[270] := B#16#0;
   FC2_RECV_1[271] := B#16#0;
   FC2_RECV_1[272] := B#16#0;
   FC2_RECV_1[273] := B#16#0;
   FC2_RECV_1[274] := B#16#0;
   FC2_RECV_1[275] := B#16#0;
   FC2_RECV_1[276] := B#16#0;
   FC2_RECV_1[277] := B#16#0;
   FC2_RECV_1[278] := B#16#0;
   FC2_RECV_1[279] := B#16#0;
   FC2_RECV_1[280] := B#16#0;
   FC2_RECV_1[281] := B#16#0;
   FC2_RECV_1[282] := B#16#0;
   FC2_RECV_1[283] := B#16#0;
   FC2_RECV_1[284] := B#16#0;
   FC2_RECV_1[285] := B#16#0;
   FC2_RECV_1[286] := B#16#0;
   FC2_RECV_1[287] := B#16#0;
   FC2_RECV_1[288] := B#16#0;
   FC2_RECV_1[289] := B#16#0;
   FC2_RECV_1[290] := B#16#0;
   FC2_RECV_1[291] := B#16#0;
   FC2_RECV_1[292] := B#16#0;
   FC2_RECV_1[293] := B#16#0;
   FC2_RECV_1[294] := B#16#0;
   FC2_RECV_1[295] := B#16#0;
   FC2_RECV_1[296] := B#16#0;
   FC2_RECV_1[297] := B#16#0;
   FC2_RECV_1[298] := B#16#0;
   FC2_RECV_1[299] := B#16#0;
   FC2_RECV_1[300] := B#16#0;
   FC2_RECV_1[301] := B#16#0;
   FC2_RECV_1[302] := B#16#0;
   FC2_RECV_1[303] := B#16#0;
   FC2_RECV_1[304] := B#16#0;
   FC2_RECV_1[305] := B#16#0;
   FC2_RECV_1[306] := B#16#0;
   FC2_RECV_1[307] := B#16#0;
   FC2_RECV_1[308] := B#16#0;
   FC2_RECV_1[309] := B#16#0;
   FC2_RECV_1[310] := B#16#0;
   FC2_RECV_1[311] := B#16#0;
   FC2_RECV_1[312] := B#16#0;
   FC2_RECV_1[313] := B#16#0;
   FC2_RECV_1[314] := B#16#0;
   FC2_RECV_1[315] := B#16#0;
   FC2_RECV_1[316] := B#16#0;
   FC2_RECV_1[317] := B#16#0;
   FC2_RECV_1[318] := B#16#0;
   FC2_RECV_1[319] := B#16#0;
   FC2_RECV_1[320] := B#16#0;
   FC2_RECV_1[321] := B#16#0;
   FC2_RECV_1[322] := B#16#0;
   FC2_RECV_1[323] := B#16#0;
   FC2_RECV_1[324] := B#16#0;
   FC2_RECV_1[325] := B#16#0;
   FC2_RECV_1[326] := B#16#0;
   FC2_RECV_1[327] := B#16#0;
   FC2_RECV_1[328] := B#16#0;
   FC2_RECV_1[329] := B#16#0;
   FC2_RECV_1[330] := B#16#0;
   FC2_RECV_1[331] := B#16#0;
   FC2_RECV_1[332] := B#16#0;
   FC2_RECV_1[333] := B#16#0;
   FC2_RECV_1[334] := B#16#0;
   FC2_RECV_1[335] := B#16#0;
   FC2_RECV_1[336] := B#16#0;
   FC2_RECV_1[337] := B#16#0;
   FC2_RECV_1[338] := B#16#0;
   FC2_RECV_1[339] := B#16#0;
   FC2_RECV_1[340] := B#16#0;
   FC2_RECV_1[341] := B#16#0;
   FC2_RECV_1[342] := B#16#0;
   FC2_RECV_1[343] := B#16#0;
   FC2_RECV_1[344] := B#16#0;
   FC2_RECV_1[345] := B#16#0;
   FC2_RECV_1[346] := B#16#0;
   FC2_RECV_1[347] := B#16#0;
   FC2_RECV_1[348] := B#16#0;
   FC2_RECV_1[349] := B#16#0;
   FC2_RECV_1[350] := B#16#0;
   FC2_RECV_1[351] := B#16#0;
   FC2_RECV_1[352] := B#16#0;
   FC2_RECV_1[353] := B#16#0;
   FC2_RECV_1[354] := B#16#0;
   FC2_RECV_1[355] := B#16#0;
   FC2_RECV_1[356] := B#16#0;
   FC2_RECV_1[357] := B#16#0;
   FC2_RECV_1[358] := B#16#0;
   FC2_RECV_1[359] := B#16#0;
   FC2_RECV_1[360] := B#16#0;
   FC2_RECV_1[361] := B#16#0;
   FC2_RECV_1[362] := B#16#0;
   FC2_RECV_1[363] := B#16#0;
   FC2_RECV_1[364] := B#16#0;
   FC2_RECV_1[365] := B#16#0;
   FC2_RECV_1[366] := B#16#0;
   FC2_RECV_1[367] := B#16#0;
   FC2_RECV_1[368] := B#16#0;
   FC2_RECV_1[369] := B#16#0;
   FC2_RECV_1[370] := B#16#0;
   FC2_RECV_1[371] := B#16#0;
   FC2_RECV_1[372] := B#16#0;
   FC2_RECV_1[373] := B#16#0;
   FC2_RECV_1[374] := B#16#0;
   FC2_RECV_1[375] := B#16#0;
   FC2_RECV_1[376] := B#16#0;
   FC2_RECV_1[377] := B#16#0;
   FC2_RECV_1[378] := B#16#0;
   FC2_RECV_1[379] := B#16#0;
   FC2_RECV_1[380] := B#16#0;
   FC2_RECV_1[381] := B#16#0;
   FC2_RECV_1[382] := B#16#0;
   FC2_RECV_1[383] := B#16#0;
   FC2_RECV_1[384] := B#16#0;
   FC2_RECV_1[385] := B#16#0;
   FC2_RECV_1[386] := B#16#0;
   FC2_RECV_1[387] := B#16#0;
   FC2_RECV_1[388] := B#16#0;
   FC2_RECV_1[389] := B#16#0;
   FC2_RECV_1[390] := B#16#0;
   FC2_RECV_1[391] := B#16#0;
   FC2_RECV_1[392] := B#16#0;
   FC2_RECV_1[393] := B#16#0;
   FC2_RECV_1[394] := B#16#0;
   FC2_RECV_1[395] := B#16#0;
   FC2_RECV_1[396] := B#16#0;
   FC2_RECV_1[397] := B#16#0;
   FC2_RECV_1[398] := B#16#0;
   FC2_RECV_1[399] := B#16#0;
   FC2_RECV_1[400] := B#16#0;
   FC2_RECV_1[401] := B#16#0;
   FC2_RECV_1[402] := B#16#0;
   FC2_RECV_1[403] := B#16#0;
   FC2_RECV_1[404] := B#16#0;
   FC2_RECV_1[405] := B#16#0;
   FC2_RECV_1[406] := B#16#0;
   FC2_RECV_1[407] := B#16#0;
   FC2_RECV_1[408] := B#16#0;
   FC2_RECV_1[409] := B#16#0;
   FC2_RECV_1[410] := B#16#0;
   FC2_RECV_1[411] := B#16#0;
   FC2_RECV_1[412] := B#16#0;
   FC2_RECV_1[413] := B#16#0;
   FC2_RECV_1[414] := B#16#0;
   FC2_RECV_1[415] := B#16#0;
   FC2_RECV_1[416] := B#16#0;
   FC2_RECV_1[417] := B#16#0;
   FC2_RECV_1[418] := B#16#0;
   FC2_RECV_1[419] := B#16#0;
   FC2_RECV_1[420] := B#16#0;
   FC2_RECV_1[421] := B#16#0;
   FC2_RECV_1[422] := B#16#0;
   FC2_RECV_1[423] := B#16#0;
   FC2_RECV_1[424] := B#16#0;
   FC2_RECV_1[425] := B#16#0;
   FC2_RECV_1[426] := B#16#0;
   FC2_RECV_1[427] := B#16#0;
   FC2_RECV_1[428] := B#16#0;
   FC2_RECV_1[429] := B#16#0;
   FC2_RECV_1[430] := B#16#0;
   FC2_RECV_1[431] := B#16#0;
   FC2_RECV_1[432] := B#16#0;
   FC2_RECV_1[433] := B#16#0;
   FC2_RECV_1[434] := B#16#0;
   FC2_RECV_1[435] := B#16#0;
   FC2_RECV_1[436] := B#16#0;
   FC2_RECV_1[437] := B#16#0;
   FC2_RECV_1[438] := B#16#0;
   FC2_RECV_1[439] := B#16#0;
   FC2_RECV_1[440] := B#16#0;
   FC2_RECV_1[441] := B#16#0;
   FC2_RECV_1[442] := B#16#0;
   FC2_RECV_1[443] := B#16#0;
   FC2_RECV_1[444] := B#16#0;
   FC2_RECV_1[445] := B#16#0;
   FC2_RECV_1[446] := B#16#0;
   FC2_RECV_1[447] := B#16#0;
   FC2_RECV_1[448] := B#16#0;
   FC2_RECV_1[449] := B#16#0;
   FC2_RECV_1[450] := B#16#0;
   FC2_RECV_1[451] := B#16#0;
   FC2_RECV_1[452] := B#16#0;
   FC2_RECV_1[453] := B#16#0;
   FC2_RECV_1[454] := B#16#0;
   FC2_RECV_1[455] := B#16#0;
   FC2_RECV_1[456] := B#16#0;
   FC2_RECV_1[457] := B#16#0;
   FC2_RECV_1[458] := B#16#0;
   FC2_RECV_1[459] := B#16#0;
   FC2_RECV_1[460] := B#16#0;
   FC2_RECV_1[461] := B#16#0;
   FC2_RECV_1[462] := B#16#0;
   FC2_RECV_1[463] := B#16#0;
   FC2_RECV_1[464] := B#16#0;
   FC2_RECV_1[465] := B#16#0;
   FC2_RECV_1[466] := B#16#0;
   FC2_RECV_1[467] := B#16#0;
   FC2_RECV_1[468] := B#16#0;
   FC2_RECV_1[469] := B#16#0;
   FC2_RECV_1[470] := B#16#0;
   FC2_RECV_1[471] := B#16#0;
   FC2_RECV_1[472] := B#16#0;
   FC2_RECV_1[473] := B#16#0;
   FC2_RECV_1[474] := B#16#0;
   FC2_RECV_1[475] := B#16#0;
   FC2_RECV_1[476] := B#16#0;
   FC2_RECV_1[477] := B#16#0;
   FC2_RECV_1[478] := B#16#0;
   FC2_RECV_1[479] := B#16#0;
   FC2_RECV_1[480] := B#16#0;
   FC2_RECV_1[481] := B#16#0;
   FC2_RECV_1[482] := B#16#0;
   FC2_RECV_1[483] := B#16#0;
   FC2_RECV_1[484] := B#16#0;
   FC2_RECV_1[485] := B#16#0;
   FC2_RECV_1[486] := B#16#0;
   FC2_RECV_1[487] := B#16#0;
   FC2_RECV_1[488] := B#16#0;
   FC2_RECV_1[489] := B#16#0;
   FC2_RECV_1[490] := B#16#0;
   FC2_RECV_1[491] := B#16#0;
   FC2_RECV_1[492] := B#16#0;
   FC2_RECV_1[493] := B#16#0;
   FC2_RECV_1[494] := B#16#0;
   FC2_RECV_1[495] := B#16#0;
   FC2_RECV_1[496] := B#16#0;
   FC2_RECV_1[497] := B#16#0;
   FC2_RECV_1[498] := B#16#0;
   FC2_RECV_1[499] := B#16#0;
   FC2_RECV_1[500] := B#16#0;
   FC2_RECV_1[501] := B#16#0;
   FC2_RECV_1[502] := B#16#0;
   FC2_RECV_1[503] := B#16#0;
   FC2_RECV_1[504] := B#16#0;
   FC2_RECV_1[505] := B#16#0;
   FC2_RECV_1[506] := B#16#0;
   FC2_RECV_1[507] := B#16#0;
   FC2_RECV_1[508] := B#16#0;
   FC2_RECV_1[509] := B#16#0;
   FC2_RECV_1[510] := B#16#0;
   FC2_RECV_1[511] := B#16#0;
   FC2_RECV_1[512] := B#16#0;
   FC2_RECV_1[513] := B#16#0;
   FC2_RECV_1[514] := B#16#0;
   FC2_RECV_1[515] := B#16#0;
   FC2_RECV_1[516] := B#16#0;
   FC2_RECV_1[517] := B#16#0;
   FC2_RECV_1[518] := B#16#0;
   FC2_RECV_1[519] := B#16#0;
   FC2_RECV_1[520] := B#16#0;
   FC2_RECV_1[521] := B#16#0;
   FC2_RECV_1[522] := B#16#0;
   FC2_RECV_1[523] := B#16#0;
   FC2_RECV_1[524] := B#16#0;
   FC2_RECV_1[525] := B#16#0;
   FC2_RECV_1[526] := B#16#0;
   FC2_RECV_1[527] := B#16#0;
   FC2_RECV_1[528] := B#16#0;
   FC2_RECV_1[529] := B#16#0;
   FC2_RECV_1[530] := B#16#0;
   FC2_RECV_1[531] := B#16#0;
   FC2_RECV_1[532] := B#16#0;
   FC2_RECV_1[533] := B#16#0;
   FC2_RECV_1[534] := B#16#0;
   FC2_RECV_1[535] := B#16#0;
   FC2_RECV_1[536] := B#16#0;
   FC2_RECV_1[537] := B#16#0;
   FC2_RECV_1[538] := B#16#0;
   FC2_RECV_1[539] := B#16#0;
   FC2_RECV_1[540] := B#16#0;
   FC2_RECV_1[541] := B#16#0;
   FC2_RECV_1[542] := B#16#0;
   FC2_RECV_1[543] := B#16#0;
   FC2_RECV_1[544] := B#16#0;
   FC2_RECV_1[545] := B#16#0;
   FC2_RECV_1[546] := B#16#0;
   FC2_RECV_1[547] := B#16#0;
   FC2_RECV_1[548] := B#16#0;
   FC2_RECV_1[549] := B#16#0;
   FC2_RECV_1[550] := B#16#0;
   FC2_RECV_1[551] := B#16#0;
   FC2_RECV_1[552] := B#16#0;
   FC2_RECV_1[553] := B#16#0;
   FC2_RECV_1[554] := B#16#0;
   FC2_RECV_1[555] := B#16#0;
   FC2_RECV_1[556] := B#16#0;
   FC2_RECV_1[557] := B#16#0;
   FC2_RECV_1[558] := B#16#0;
   FC2_RECV_1[559] := B#16#0;
   FC2_RECV_1[560] := B#16#0;
   FC2_RECV_1[561] := B#16#0;
   FC2_RECV_1[562] := B#16#0;
   FC2_RECV_1[563] := B#16#0;
   FC2_RECV_1[564] := B#16#0;
   FC2_RECV_1[565] := B#16#0;
   FC2_RECV_1[566] := B#16#0;
   FC2_RECV_1[567] := B#16#0;
   FC2_RECV_1[568] := B#16#0;
   FC2_RECV_1[569] := B#16#0;
   FC2_RECV_1[570] := B#16#0;
   FC2_RECV_1[571] := B#16#0;
   FC2_RECV_1[572] := B#16#0;
   FC2_RECV_1[573] := B#16#0;
   FC2_RECV_1[574] := B#16#0;
   FC2_RECV_1[575] := B#16#0;
   FC2_RECV_1[576] := B#16#0;
   FC2_RECV_1[577] := B#16#0;
   FC2_RECV_1[578] := B#16#0;
   FC2_RECV_1[579] := B#16#0;
   FC2_RECV_1[580] := B#16#0;
   FC2_RECV_1[581] := B#16#0;
   FC2_RECV_1[582] := B#16#0;
   FC2_RECV_1[583] := B#16#0;
   FC2_RECV_1[584] := B#16#0;
   FC2_RECV_1[585] := B#16#0;
   FC2_RECV_1[586] := B#16#0;
   FC2_RECV_1[587] := B#16#0;
   FC2_RECV_1[588] := B#16#0;
   FC2_RECV_1[589] := B#16#0;
   FC2_RECV_1[590] := B#16#0;
   FC2_RECV_1[591] := B#16#0;
   FC2_RECV_1[592] := B#16#0;
   FC2_RECV_1[593] := B#16#0;
   FC2_RECV_1[594] := B#16#0;
   FC2_RECV_1[595] := B#16#0;
   FC2_RECV_1[596] := B#16#0;
   FC2_RECV_1[597] := B#16#0;
   FC2_RECV_1[598] := B#16#0;
   FC2_RECV_1[599] := B#16#0;
   FC2_RECV_1[600] := B#16#0;
   FC2_RECV_1[601] := B#16#0;
   FC2_RECV_1[602] := B#16#0;
   FC2_RECV_1[603] := B#16#0;
   FC2_RECV_1[604] := B#16#0;
   FC2_RECV_1[605] := B#16#0;
   FC2_RECV_1[606] := B#16#0;
   FC2_RECV_1[607] := B#16#0;
   FC2_RECV_1[608] := B#16#0;
   FC2_RECV_1[609] := B#16#0;
   FC2_RECV_1[610] := B#16#0;
   FC2_RECV_1[611] := B#16#0;
   FC2_RECV_1[612] := B#16#0;
   FC2_RECV_1[613] := B#16#0;
   FC2_RECV_1[614] := B#16#0;
   FC2_RECV_1[615] := B#16#0;
   FC2_RECV_1[616] := B#16#0;
   FC2_RECV_1[617] := B#16#0;
   FC2_RECV_1[618] := B#16#0;
   FC2_RECV_1[619] := B#16#0;
   FC2_RECV_1[620] := B#16#0;
   FC2_RECV_1[621] := B#16#0;
   FC2_RECV_1[622] := B#16#0;
   FC2_RECV_1[623] := B#16#0;
   FC2_RECV_1[624] := B#16#0;
   FC2_RECV_1[625] := B#16#0;
   FC2_RECV_1[626] := B#16#0;
   FC2_RECV_1[627] := B#16#0;
   FC2_RECV_1[628] := B#16#0;
   FC2_RECV_1[629] := B#16#0;
   FC2_RECV_1[630] := B#16#0;
   FC2_RECV_1[631] := B#16#0;
   FC2_RECV_1[632] := B#16#0;
   FC2_RECV_1[633] := B#16#0;
   FC2_RECV_1[634] := B#16#0;
   FC2_RECV_1[635] := B#16#0;
   FC2_RECV_1[636] := B#16#0;
   FC2_RECV_1[637] := B#16#0;
   FC2_RECV_1[638] := B#16#0;
   FC2_RECV_1[639] := B#16#0;
   FC2_RECV_1[640] := B#16#0;
   FC2_RECV_1[641] := B#16#0;
   FC2_RECV_1[642] := B#16#0;
   FC2_RECV_1[643] := B#16#0;
   FC2_RECV_1[644] := B#16#0;
   FC2_RECV_1[645] := B#16#0;
   FC2_RECV_1[646] := B#16#0;
   FC2_RECV_1[647] := B#16#0;
   FC2_RECV_1[648] := B#16#0;
   FC2_RECV_1[649] := B#16#0;
   FC2_RECV_1[650] := B#16#0;
   FC2_RECV_1[651] := B#16#0;
   FC2_RECV_1[652] := B#16#0;
   FC2_RECV_1[653] := B#16#0;
   FC2_RECV_1[654] := B#16#0;
   FC2_RECV_1[655] := B#16#0;
   FC2_RECV_1[656] := B#16#0;
   FC2_RECV_1[657] := B#16#0;
   FC2_RECV_1[658] := B#16#0;
   FC2_RECV_1[659] := B#16#0;
   FC2_RECV_1[660] := B#16#0;
   FC2_RECV_1[661] := B#16#0;
   FC2_RECV_1[662] := B#16#0;
   FC2_RECV_1[663] := B#16#0;
   FC2_RECV_1[664] := B#16#0;
   FC2_RECV_1[665] := B#16#0;
   FC2_RECV_1[666] := B#16#0;
   FC2_RECV_1[667] := B#16#0;
   FC2_RECV_1[668] := B#16#0;
   FC2_RECV_1[669] := B#16#0;
   FC2_RECV_1[670] := B#16#0;
   FC2_RECV_1[671] := B#16#0;
   FC2_RECV_1[672] := B#16#0;
   FC2_RECV_1[673] := B#16#0;
   FC2_RECV_1[674] := B#16#0;
   FC2_RECV_1[675] := B#16#0;
   FC2_RECV_1[676] := B#16#0;
   FC2_RECV_1[677] := B#16#0;
   FC2_RECV_1[678] := B#16#0;
   FC2_RECV_1[679] := B#16#0;
   FC2_RECV_1[680] := B#16#0;
   FC2_RECV_1[681] := B#16#0;
   FC2_RECV_1[682] := B#16#0;
   FC2_RECV_1[683] := B#16#0;
   FC2_RECV_1[684] := B#16#0;
   FC2_RECV_1[685] := B#16#0;
   FC2_RECV_1[686] := B#16#0;
   FC2_RECV_1[687] := B#16#0;
   FC2_RECV_1[688] := B#16#0;
   FC2_RECV_1[689] := B#16#0;
   FC2_RECV_1[690] := B#16#0;
   FC2_RECV_1[691] := B#16#0;
   FC2_RECV_1[692] := B#16#0;
   FC2_RECV_1[693] := B#16#0;
   FC2_RECV_1[694] := B#16#0;
   FC2_RECV_1[695] := B#16#0;
   FC2_RECV_1[696] := B#16#0;
   FC2_RECV_1[697] := B#16#0;
   FC2_RECV_1[698] := B#16#0;
   FC2_RECV_1[699] := B#16#0;
END_DATA_BLOCK

DATA_BLOCK DB 98
VERSION : 0.1


  STRUCT
   STAT0 : ARRAY  [0 .. 25 ] OF DWORD ;
  END_STRUCT ;
BEGIN
   STAT0[0] := DW#16#0;
   STAT0[1] := DW#16#0;
   STAT0[2] := DW#16#0;
   STAT0[3] := DW#16#0;
   STAT0[4] := DW#16#0;
   STAT0[5] := DW#16#0;
   STAT0[6] := DW#16#0;
   STAT0[7] := DW#16#0;
   STAT0[8] := DW#16#0;
   STAT0[9] := DW#16#0;
   STAT0[10] := DW#16#0;
   STAT0[11] := DW#16#0;
   STAT0[12] := DW#16#0;
   STAT0[13] := DW#16#0;
   STAT0[14] := DW#16#0;
   STAT0[15] := DW#16#0;
   STAT0[16] := DW#16#0;
   STAT0[17] := DW#16#0;
   STAT0[18] := DW#16#0;
   STAT0[19] := DW#16#0;
   STAT0[20] := DW#16#0;
   STAT0[21] := DW#16#0;
   STAT0[22] := DW#16#0;
   STAT0[23] := DW#16#0;
   STAT0[24] := DW#16#0;
   STAT0[25] := DW#16#0;
END_DATA_BLOCK

DATA_BLOCK DB 100
TITLE =
VERSION : 0.1


  STRUCT
   STN1_KEY : UDT 1;
   STN2_RB : UDT 1;
   STN3_IDLE : UDT 1;
   FA_BT : UDT 1;
  END_STRUCT ;
BEGIN
   STN1_KEY.VIN_NO_1 := B#16#0;
   STN1_KEY.VIN_NO_2 := B#16#0;
   STN1_KEY.VIN_NO_3 := B#16#0;
   STN1_KEY.VIN_NO_SP := B#16#0;
   STN1_KEY.BT1_TL := FALSE;
   STN1_KEY.BT1_LM := TRUE;
   STN1_KEY.BT1_EF := FALSE;
   STN1_KEY.SP1 := FALSE;
   STN1_KEY.SP2 := FALSE;
   STN1_KEY.BT2_5P := FALSE;
   STN1_KEY.BT2_7P := TRUE;
   STN1_KEY.SP3 := FALSE;
   STN1_KEY.SP4 := FALSE;
   STN1_KEY.BT3_LHD := TRUE;
   STN1_KEY.BT3_RHD := FALSE;
   STN1_KEY.BT4_DOM := FALSE;
   STN1_KEY.BT4_EXP := FALSE;
   STN1_KEY.BT4_NAS := TRUE;
   STN1_KEY.BT4_EEC := FALSE;
   STN1_KEY.BT4_AUS := FALSE;
   STN1_KEY.BT4_BRJ := FALSE;
   STN1_KEY.BT4_ME := FALSE;
   STN1_KEY.BT4_JAP := FALSE;
   STN1_KEY.BT4_IND := FALSE;
   STN1_KEY.SP5 := FALSE;
   STN1_KEY.SP6 := FALSE;
   STN1_KEY.BT5_CR := FALSE;
   STN1_KEY.BT5_GA := TRUE;
   STN1_KEY.BT6_35_GSL := FALSE;
   STN1_KEY.BT6_27_GSL := TRUE;
   STN1_KEY.BT6_20_GSL := FALSE;
   STN1_KEY.BT6_29_DSL := FALSE;
   STN1_KEY.BT6_20_DSL := FALSE;
   STN1_KEY.BT6_25_DSL := FALSE;
   STN1_KEY.SP7 := FALSE;
   STN1_KEY.BT6_LMFC := FALSE;
   STN1_KEY.BT7_MT := FALSE;
   STN1_KEY.BT7_AT := TRUE;
   STN1_KEY.BT8_G_ROOF := TRUE;
   STN1_KEY.BT8_S_ROOF := FALSE;
   STN1_KEY.BT9_2WD := TRUE;
   STN1_KEY.BT9_4WD := FALSE;
   STN1_KEY.BT10_PROOF := FALSE;
   STN1_KEY.SP10 := FALSE;
   STN1_KEY.BT11_MTS := FALSE;
   STN1_KEY.BT11_S_LAMP := FALSE;
   STN1_KEY.BT11_GARNISH := FALSE;
   STN1_KEY.BT11_HMSL := FALSE;
   STN1_KEY.BT11_ABS := FALSE;
   STN1_KEY.BT11_AV := FALSE;
   STN1_KEY.BT11_RACK := FALSE;
   STN1_KEY.BT11_S_HOLD := FALSE;
   STN1_KEY.BT11_SPOILER := FALSE;
   STN1_KEY.BT11_W_NOZZLE := FALSE;
   STN1_KEY.BT11_U_MIRROR := FALSE;
   STN1_KEY.BT11_P_ANT := FALSE;
   STN1_KEY.BT11_A_CLEAN := FALSE;
   STN1_KEY.SP11 := FALSE;
   STN1_KEY.SP12 := FALSE;
   STN1_KEY.SP13 := FALSE;
   STN1_KEY.SP14 := FALSE;
   STN1_KEY.SP15 := FALSE;
   STN1_KEY.BT12_VAC := FALSE;
   STN1_KEY.BT12_NG_CAR := FALSE;
   STN1_KEY.BT12_NG_FLATCAR := FALSE;
   STN1_KEY.BT12_UNLOADING := FALSE;
   STN1_KEY.BT12_AS := FALSE;
   STN1_KEY.SP16 := FALSE;
   STN1_KEY.SP_WORD_1 := B#16#0;
   STN1_KEY.SP_WORD_2 := B#16#0;
   STN1_KEY.SP_WORD_3 := B#16#0;
   STN1_KEY.SP_WORD_4 := B#16#0;
   STN1_KEY.AUX_BIT[1] := TRUE;
   STN1_KEY.AUX_BIT[2] := FALSE;
   STN1_KEY.AUX_BIT[3] := FALSE;
   STN1_KEY.AUX_BIT[4] := FALSE;
   STN1_KEY.AUX_BIT[5] := FALSE;
   STN1_KEY.AUX_BIT[6] := FALSE;
   STN1_KEY.AUX_BIT[7] := FALSE;
   STN1_KEY.AUX_BIT[8] := FALSE;
   STN1_KEY.AUX_BIT[9] := FALSE;
   STN1_KEY.AUX_BIT[10] := FALSE;
   STN1_KEY.AUX_BIT[11] := FALSE;
   STN1_KEY.AUX_BIT[12] := FALSE;
   STN1_KEY.AUX_BIT[13] := FALSE;
   STN1_KEY.AUX_BIT[14] := FALSE;
   STN1_KEY.AUX_BIT[15] := FALSE;
   STN1_KEY.AUX_BIT[16] := FALSE;
   STN1_KEY.AUX_BIT[17] := FALSE;
   STN1_KEY.AUX_BIT[18] := FALSE;
   STN1_KEY.AUX_BIT[19] := FALSE;
   STN1_KEY.AUX_BIT[20] := FALSE;
   STN1_KEY.AUX_BIT[21] := FALSE;
   STN1_KEY.AUX_BIT[22] := FALSE;
   STN1_KEY.AUX_BIT[23] := FALSE;
   STN1_KEY.AUX_BIT[24] := FALSE;
   STN1_KEY.AUX_BIT[25] := FALSE;
   STN1_KEY.AUX_BIT[26] := FALSE;
   STN1_KEY.AUX_BIT[27] := FALSE;
   STN1_KEY.AUX_BIT[28] := FALSE;
   STN1_KEY.AUX_BIT[29] := FALSE;
   STN1_KEY.AUX_BIT[30] := FALSE;
   STN1_KEY.AUX_BIT[31] := FALSE;
   STN1_KEY.AUX_BIT[32] := FALSE;
   STN2_RB.VIN_NO_1 := B#16#0;
   STN2_RB.VIN_NO_2 := B#16#0;
   STN2_RB.VIN_NO_3 := B#16#0;
   STN2_RB.VIN_NO_SP := B#16#0;
   STN2_RB.BT1_TL := FALSE;
   STN2_RB.BT1_LM := FALSE;
   STN2_RB.BT1_EF := FALSE;
   STN2_RB.SP1 := FALSE;
   STN2_RB.SP2 := FALSE;
   STN2_RB.BT2_5P := FALSE;
   STN2_RB.BT2_7P := FALSE;
   STN2_RB.SP3 := FALSE;
   STN2_RB.SP4 := FALSE;
   STN2_RB.BT3_LHD := FALSE;
   STN2_RB.BT3_RHD := FALSE;
   STN2_RB.BT4_DOM := FALSE;
   STN2_RB.BT4_EXP := FALSE;
   STN2_RB.BT4_NAS := FALSE;
   STN2_RB.BT4_EEC := FALSE;
   STN2_RB.BT4_AUS := FALSE;
   STN2_RB.BT4_BRJ := FALSE;
   STN2_RB.BT4_ME := FALSE;
   STN2_RB.BT4_JAP := FALSE;
   STN2_RB.BT4_IND := FALSE;
   STN2_RB.SP5 := FALSE;
   STN2_RB.SP6 := FALSE;
   STN2_RB.BT5_CR := FALSE;
   STN2_RB.BT5_GA := FALSE;
   STN2_RB.BT6_35_GSL := FALSE;
   STN2_RB.BT6_27_GSL := FALSE;
   STN2_RB.BT6_20_GSL := FALSE;
   STN2_RB.BT6_29_DSL := FALSE;
   STN2_RB.BT6_20_DSL := FALSE;
   STN2_RB.BT6_25_DSL := FALSE;
   STN2_RB.SP7 := FALSE;
   STN2_RB.BT6_LMFC := FALSE;
   STN2_RB.BT7_MT := FALSE;
   STN2_RB.BT7_AT := FALSE;
   STN2_RB.BT8_G_ROOF := FALSE;
   STN2_RB.BT8_S_ROOF := FALSE;
   STN2_RB.BT9_2WD := FALSE;
   STN2_RB.BT9_4WD := FALSE;
   STN2_RB.BT10_PROOF := FALSE;
   STN2_RB.SP10 := FALSE;
   STN2_RB.BT11_MTS := FALSE;
   STN2_RB.BT11_S_LAMP := FALSE;
   STN2_RB.BT11_GARNISH := FALSE;
   STN2_RB.BT11_HMSL := FALSE;
   STN2_RB.BT11_ABS := FALSE;
   STN2_RB.BT11_AV := FALSE;
   STN2_RB.BT11_RACK := FALSE;
   STN2_RB.BT11_S_HOLD := FALSE;
   STN2_RB.BT11_SPOILER := FALSE;
   STN2_RB.BT11_W_NOZZLE := FALSE;
   STN2_RB.BT11_U_MIRROR := FALSE;
   STN2_RB.BT11_P_ANT := FALSE;
   STN2_RB.BT11_A_CLEAN := FALSE;
   STN2_RB.SP11 := FALSE;
   STN2_RB.SP12 := FALSE;
   STN2_RB.SP13 := FALSE;
   STN2_RB.SP14 := FALSE;
   STN2_RB.SP15 := FALSE;
   STN2_RB.BT12_VAC := FALSE;
   STN2_RB.BT12_NG_CAR := FALSE;
   STN2_RB.BT12_NG_FLATCAR := FALSE;
   STN2_RB.BT12_UNLOADING := FALSE;
   STN2_RB.BT12_AS := FALSE;
   STN2_RB.SP16 := FALSE;
   STN2_RB.SP_WORD_1 := B#16#0;
   STN2_RB.SP_WORD_2 := B#16#0;
   STN2_RB.SP_WORD_3 := B#16#0;
   STN2_RB.SP_WORD_4 := B#16#0;
   STN2_RB.AUX_BIT[1] := FALSE;
   STN2_RB.AUX_BIT[2] := FALSE;
   STN2_RB.AUX_BIT[3] := FALSE;
   STN2_RB.AUX_BIT[4] := FALSE;
   STN2_RB.AUX_BIT[5] := FALSE;
   STN2_RB.AUX_BIT[6] := FALSE;
   STN2_RB.AUX_BIT[7] := FALSE;
   STN2_RB.AUX_BIT[8] := FALSE;
   STN2_RB.AUX_BIT[9] := FALSE;
   STN2_RB.AUX_BIT[10] := FALSE;
   STN2_RB.AUX_BIT[11] := FALSE;
   STN2_RB.AUX_BIT[12] := FALSE;
   STN2_RB.AUX_BIT[13] := FALSE;
   STN2_RB.AUX_BIT[14] := FALSE;
   STN2_RB.AUX_BIT[15] := FALSE;
   STN2_RB.AUX_BIT[16] := FALSE;
   STN2_RB.AUX_BIT[17] := FALSE;
   STN2_RB.AUX_BIT[18] := FALSE;
   STN2_RB.AUX_BIT[19] := FALSE;
   STN2_RB.AUX_BIT[20] := FALSE;
   STN2_RB.AUX_BIT[21] := FALSE;
   STN2_RB.AUX_BIT[22] := FALSE;
   STN2_RB.AUX_BIT[23] := FALSE;
   STN2_RB.AUX_BIT[24] := FALSE;
   STN2_RB.AUX_BIT[25] := FALSE;
   STN2_RB.AUX_BIT[26] := FALSE;
   STN2_RB.AUX_BIT[27] := FALSE;
   STN2_RB.AUX_BIT[28] := FALSE;
   STN2_RB.AUX_BIT[29] := FALSE;
   STN2_RB.AUX_BIT[30] := FALSE;
   STN2_RB.AUX_BIT[31] := FALSE;
   STN2_RB.AUX_BIT[32] := FALSE;
   STN3_IDLE.VIN_NO_1 := B#16#0;
   STN3_IDLE.VIN_NO_2 := B#16#0;
   STN3_IDLE.VIN_NO_3 := B#16#0;
   STN3_IDLE.VIN_NO_SP := B#16#0;
   STN3_IDLE.BT1_TL := FALSE;
   STN3_IDLE.BT1_LM := TRUE;
   STN3_IDLE.BT1_EF := FALSE;
   STN3_IDLE.SP1 := FALSE;
   STN3_IDLE.SP2 := FALSE;
   STN3_IDLE.BT2_5P := FALSE;
   STN3_IDLE.BT2_7P := TRUE;
   STN3_IDLE.SP3 := FALSE;
   STN3_IDLE.SP4 := FALSE;
   STN3_IDLE.BT3_LHD := TRUE;
   STN3_IDLE.BT3_RHD := FALSE;
   STN3_IDLE.BT4_DOM := FALSE;
   STN3_IDLE.BT4_EXP := FALSE;
   STN3_IDLE.BT4_NAS := TRUE;
   STN3_IDLE.BT4_EEC := FALSE;
   STN3_IDLE.BT4_AUS := FALSE;
   STN3_IDLE.BT4_BRJ := FALSE;
   STN3_IDLE.BT4_ME := FALSE;
   STN3_IDLE.BT4_JAP := FALSE;
   STN3_IDLE.BT4_IND := FALSE;
   STN3_IDLE.SP5 := FALSE;
   STN3_IDLE.SP6 := FALSE;
   STN3_IDLE.BT5_CR := FALSE;
   STN3_IDLE.BT5_GA := TRUE;
   STN3_IDLE.BT6_35_GSL := FALSE;
   STN3_IDLE.BT6_27_GSL := TRUE;
   STN3_IDLE.BT6_20_GSL := FALSE;
   STN3_IDLE.BT6_29_DSL := FALSE;
   STN3_IDLE.BT6_20_DSL := FALSE;
   STN3_IDLE.BT6_25_DSL := FALSE;
   STN3_IDLE.SP7 := FALSE;
   STN3_IDLE.BT6_LMFC := FALSE;
   STN3_IDLE.BT7_MT := FALSE;
   STN3_IDLE.BT7_AT := TRUE;
   STN3_IDLE.BT8_G_ROOF := TRUE;
   STN3_IDLE.BT8_S_ROOF := FALSE;
   STN3_IDLE.BT9_2WD := TRUE;
   STN3_IDLE.BT9_4WD := FALSE;
   STN3_IDLE.BT10_PROOF := FALSE;
   STN3_IDLE.SP10 := FALSE;
   STN3_IDLE.BT11_MTS := FALSE;
   STN3_IDLE.BT11_S_LAMP := FALSE;
   STN3_IDLE.BT11_GARNISH := FALSE;
   STN3_IDLE.BT11_HMSL := FALSE;
   STN3_IDLE.BT11_ABS := FALSE;
   STN3_IDLE.BT11_AV := FALSE;
   STN3_IDLE.BT11_RACK := FALSE;
   STN3_IDLE.BT11_S_HOLD := FALSE;
   STN3_IDLE.BT11_SPOILER := FALSE;
   STN3_IDLE.BT11_W_NOZZLE := FALSE;
   STN3_IDLE.BT11_U_MIRROR := FALSE;
   STN3_IDLE.BT11_P_ANT := FALSE;
   STN3_IDLE.BT11_A_CLEAN := FALSE;
   STN3_IDLE.SP11 := FALSE;
   STN3_IDLE.SP12 := FALSE;
   STN3_IDLE.SP13 := FALSE;
   STN3_IDLE.SP14 := FALSE;
   STN3_IDLE.SP15 := FALSE;
   STN3_IDLE.BT12_VAC := FALSE;
   STN3_IDLE.BT12_NG_CAR := FALSE;
   STN3_IDLE.BT12_NG_FLATCAR := FALSE;
   STN3_IDLE.BT12_UNLOADING := FALSE;
   STN3_IDLE.BT12_AS := FALSE;
   STN3_IDLE.SP16 := FALSE;
   STN3_IDLE.SP_WORD_1 := B#16#0;
   STN3_IDLE.SP_WORD_2 := B#16#0;
   STN3_IDLE.SP_WORD_3 := B#16#0;
   STN3_IDLE.SP_WORD_4 := B#16#0;
   STN3_IDLE.AUX_BIT[1] := FALSE;
   STN3_IDLE.AUX_BIT[2] := FALSE;
   STN3_IDLE.AUX_BIT[3] := FALSE;
   STN3_IDLE.AUX_BIT[4] := FALSE;
   STN3_IDLE.AUX_BIT[5] := FALSE;
   STN3_IDLE.AUX_BIT[6] := FALSE;
   STN3_IDLE.AUX_BIT[7] := FALSE;
   STN3_IDLE.AUX_BIT[8] := FALSE;
   STN3_IDLE.AUX_BIT[9] := FALSE;
   STN3_IDLE.AUX_BIT[10] := FALSE;
   STN3_IDLE.AUX_BIT[11] := FALSE;
   STN3_IDLE.AUX_BIT[12] := FALSE;
   STN3_IDLE.AUX_BIT[13] := FALSE;
   STN3_IDLE.AUX_BIT[14] := FALSE;
   STN3_IDLE.AUX_BIT[15] := FALSE;
   STN3_IDLE.AUX_BIT[16] := FALSE;
   STN3_IDLE.AUX_BIT[17] := FALSE;
   STN3_IDLE.AUX_BIT[18] := FALSE;
   STN3_IDLE.AUX_BIT[19] := FALSE;
   STN3_IDLE.AUX_BIT[20] := FALSE;
   STN3_IDLE.AUX_BIT[21] := FALSE;
   STN3_IDLE.AUX_BIT[22] := FALSE;
   STN3_IDLE.AUX_BIT[23] := FALSE;
   STN3_IDLE.AUX_BIT[24] := FALSE;
   STN3_IDLE.AUX_BIT[25] := FALSE;
   STN3_IDLE.AUX_BIT[26] := FALSE;
   STN3_IDLE.AUX_BIT[27] := FALSE;
   STN3_IDLE.AUX_BIT[28] := FALSE;
   STN3_IDLE.AUX_BIT[29] := FALSE;
   STN3_IDLE.AUX_BIT[30] := FALSE;
   STN3_IDLE.AUX_BIT[31] := FALSE;
   STN3_IDLE.AUX_BIT[32] := FALSE;
   FA_BT.VIN_NO_1 := B#16#0;
   FA_BT.VIN_NO_2 := B#16#0;
   FA_BT.VIN_NO_3 := B#16#0;
   FA_BT.VIN_NO_SP := B#16#0;
   FA_BT.BT1_TL := FALSE;
   FA_BT.BT1_LM := FALSE;
   FA_BT.BT1_EF := FALSE;
   FA_BT.SP1 := FALSE;
   FA_BT.SP2 := FALSE;
   FA_BT.BT2_5P := FALSE;
   FA_BT.BT2_7P := FALSE;
   FA_BT.SP3 := FALSE;
   FA_BT.SP4 := FALSE;
   FA_BT.BT3_LHD := FALSE;
   FA_BT.BT3_RHD := FALSE;
   FA_BT.BT4_DOM := FALSE;
   FA_BT.BT4_EXP := FALSE;
   FA_BT.BT4_NAS := FALSE;
   FA_BT.BT4_EEC := FALSE;
   FA_BT.BT4_AUS := FALSE;
   FA_BT.BT4_BRJ := FALSE;
   FA_BT.BT4_ME := FALSE;
   FA_BT.BT4_JAP := FALSE;
   FA_BT.BT4_IND := FALSE;
   FA_BT.SP5 := FALSE;
   FA_BT.SP6 := FALSE;
   FA_BT.BT5_CR := FALSE;
   FA_BT.BT5_GA := FALSE;
   FA_BT.BT6_35_GSL := FALSE;
   FA_BT.BT6_27_GSL := FALSE;
   FA_BT.BT6_20_GSL := FALSE;
   FA_BT.BT6_29_DSL := FALSE;
   FA_BT.BT6_20_DSL := FALSE;
   FA_BT.BT6_25_DSL := FALSE;
   FA_BT.SP7 := FALSE;
   FA_BT.BT6_LMFC := FALSE;
   FA_BT.BT7_MT := FALSE;
   FA_BT.BT7_AT := FALSE;
   FA_BT.BT8_G_ROOF := FALSE;
   FA_BT.BT8_S_ROOF := FALSE;
   FA_BT.BT9_2WD := FALSE;
   FA_BT.BT9_4WD := FALSE;
   FA_BT.BT10_PROOF := FALSE;
   FA_BT.SP10 := FALSE;
   FA_BT.BT11_MTS := FALSE;
   FA_BT.BT11_S_LAMP := FALSE;
   FA_BT.BT11_GARNISH := FALSE;
   FA_BT.BT11_HMSL := FALSE;
   FA_BT.BT11_ABS := FALSE;
   FA_BT.BT11_AV := FALSE;
   FA_BT.BT11_RACK := FALSE;
   FA_BT.BT11_S_HOLD := FALSE;
   FA_BT.BT11_SPOILER := FALSE;
   FA_BT.BT11_W_NOZZLE := FALSE;
   FA_BT.BT11_U_MIRROR := FALSE;
   FA_BT.BT11_P_ANT := FALSE;
   FA_BT.BT11_A_CLEAN := FALSE;
   FA_BT.SP11 := FALSE;
   FA_BT.SP12 := FALSE;
   FA_BT.SP13 := FALSE;
   FA_BT.SP14 := FALSE;
   FA_BT.SP15 := FALSE;
   FA_BT.BT12_VAC := FALSE;
   FA_BT.BT12_NG_CAR := FALSE;
   FA_BT.BT12_NG_FLATCAR := FALSE;
   FA_BT.BT12_UNLOADING := FALSE;
   FA_BT.BT12_AS := FALSE;
   FA_BT.SP16 := FALSE;
   FA_BT.SP_WORD_1 := B#16#0;
   FA_BT.SP_WORD_2 := B#16#0;
   FA_BT.SP_WORD_3 := B#16#0;
   FA_BT.SP_WORD_4 := B#16#0;
   FA_BT.AUX_BIT[1] := FALSE;
   FA_BT.AUX_BIT[2] := FALSE;
   FA_BT.AUX_BIT[3] := FALSE;
   FA_BT.AUX_BIT[4] := FALSE;
   FA_BT.AUX_BIT[5] := FALSE;
   FA_BT.AUX_BIT[6] := FALSE;
   FA_BT.AUX_BIT[7] := FALSE;
   FA_BT.AUX_BIT[8] := FALSE;
   FA_BT.AUX_BIT[9] := FALSE;
   FA_BT.AUX_BIT[10] := FALSE;
   FA_BT.AUX_BIT[11] := FALSE;
   FA_BT.AUX_BIT[12] := FALSE;
   FA_BT.AUX_BIT[13] := FALSE;
   FA_BT.AUX_BIT[14] := FALSE;
   FA_BT.AUX_BIT[15] := FALSE;
   FA_BT.AUX_BIT[16] := FALSE;
   FA_BT.AUX_BIT[17] := FALSE;
   FA_BT.AUX_BIT[18] := FALSE;
   FA_BT.AUX_BIT[19] := FALSE;
   FA_BT.AUX_BIT[20] := FALSE;
   FA_BT.AUX_BIT[21] := FALSE;
   FA_BT.AUX_BIT[22] := FALSE;
   FA_BT.AUX_BIT[23] := FALSE;
   FA_BT.AUX_BIT[24] := FALSE;
   FA_BT.AUX_BIT[25] := FALSE;
   FA_BT.AUX_BIT[26] := FALSE;
   FA_BT.AUX_BIT[27] := FALSE;
   FA_BT.AUX_BIT[28] := FALSE;
   FA_BT.AUX_BIT[29] := FALSE;
   FA_BT.AUX_BIT[30] := FALSE;
   FA_BT.AUX_BIT[31] := FALSE;
   FA_BT.AUX_BIT[32] := FALSE;
END_DATA_BLOCK

DATA_BLOCK DB 130
TITLE =
VERSION : 0.1


  STRUCT
   STAT0 : ARRAY  [0 .. 99 ] OF BYTE ;
  END_STRUCT ;
BEGIN
   STAT0[0] := B#16#2D;
   STAT0[1] := B#16#3;
   STAT0[2] := B#16#0;
   STAT0[3] := B#16#0;
   STAT0[4] := B#16#0;
   STAT0[5] := B#16#0;
   STAT0[6] := B#16#0;
   STAT0[7] := B#16#0;
   STAT0[8] := B#16#24;
   STAT0[9] := B#16#0;
   STAT0[10] := B#16#0;
   STAT0[11] := B#16#0;
   STAT0[12] := B#16#0;
   STAT0[13] := B#16#0;
   STAT0[14] := B#16#0;
   STAT0[15] := B#16#0;
   STAT0[16] := B#16#0;
   STAT0[17] := B#16#0;
   STAT0[18] := B#16#0;
   STAT0[19] := B#16#0;
   STAT0[20] := B#16#0;
   STAT0[21] := B#16#0;
   STAT0[22] := B#16#0;
   STAT0[23] := B#16#0;
   STAT0[24] := B#16#0;
   STAT0[25] := B#16#0;
   STAT0[26] := B#16#0;
   STAT0[27] := B#16#0;
   STAT0[28] := B#16#0;
   STAT0[29] := B#16#0;
   STAT0[30] := B#16#0;
   STAT0[31] := B#16#0;
   STAT0[32] := B#16#0;
   STAT0[33] := B#16#0;
   STAT0[34] := B#16#0;
   STAT0[35] := B#16#0;
   STAT0[36] := B#16#0;
   STAT0[37] := B#16#0;
   STAT0[38] := B#16#0;
   STAT0[39] := B#16#0;
   STAT0[40] := B#16#0;
   STAT0[41] := B#16#0;
   STAT0[42] := B#16#0;
   STAT0[43] := B#16#0;
   STAT0[44] := B#16#0;
   STAT0[45] := B#16#0;
   STAT0[46] := B#16#0;
   STAT0[47] := B#16#0;
   STAT0[48] := B#16#0;
   STAT0[49] := B#16#0;
   STAT0[50] := B#16#0;
   STAT0[51] := B#16#0;
   STAT0[52] := B#16#0;
   STAT0[53] := B#16#0;
   STAT0[54] := B#16#0;
   STAT0[55] := B#16#0;
   STAT0[56] := B#16#0;
   STAT0[57] := B#16#0;
   STAT0[58] := B#16#0;
   STAT0[59] := B#16#0;
   STAT0[60] := B#16#0;
   STAT0[61] := B#16#0;
   STAT0[62] := B#16#0;
   STAT0[63] := B#16#0;
   STAT0[64] := B#16#0;
   STAT0[65] := B#16#0;
   STAT0[66] := B#16#0;
   STAT0[67] := B#16#0;
   STAT0[68] := B#16#0;
   STAT0[69] := B#16#0;
   STAT0[70] := B#16#0;
   STAT0[71] := B#16#0;
   STAT0[72] := B#16#0;
   STAT0[73] := B#16#0;
   STAT0[74] := B#16#0;
   STAT0[75] := B#16#0;
   STAT0[76] := B#16#0;
   STAT0[77] := B#16#0;
   STAT0[78] := B#16#0;
   STAT0[79] := B#16#0;
   STAT0[80] := B#16#0;
   STAT0[81] := B#16#0;
   STAT0[82] := B#16#0;
   STAT0[83] := B#16#0;
   STAT0[84] := B#16#0;
   STAT0[85] := B#16#0;
   STAT0[86] := B#16#0;
   STAT0[87] := B#16#0;
   STAT0[88] := B#16#0;
   STAT0[89] := B#16#0;
   STAT0[90] := B#16#0;
   STAT0[91] := B#16#0;
   STAT0[92] := B#16#0;
   STAT0[93] := B#16#0;
   STAT0[94] := B#16#0;
   STAT0[95] := B#16#0;
   STAT0[96] := B#16#0;
   STAT0[97] := B#16#0;
   STAT0[98] := B#16#0;
   STAT0[99] := B#16#0;
END_DATA_BLOCK

DATA_BLOCK DB 160
TITLE =
VERSION : 0.1


